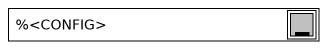
[picture p166: DIGOUT_TOUCH_SMAL (HMI screen)]
rectangle at (0,0)-(311,33): taps $Station$.$Output$
rounded rectangle at (1,1)-(280,32): text "%<CONFIG>"; shows '$Output$'; taps $Station$.$Output$; dynamic style $OutputLocked$
rounded rectangle at (279,2)-(308,31): alarm colour if $OutputLocked$; taps $Station$.$Output$; dynamic style $OutputLocked$
rounded rectangle at (282,5)-(305,28): alarm colour if $Station$.$Output$; taps $Station$.$Output$; tooltip $Output$; dynamic style $OutputLocked$
rectangle at (287,24)-(301,28): invisible if $Station$.$Output$; taps $Station$.$Output$; dynamic style gi16_betriebsart <> HAND
*)

(* Visualisation PRUEFTEILEN_CZ
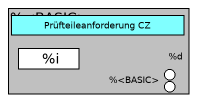
rectangle at (0,0)-(181,86): text "%<BASIC>"; shows 'auto_Prüfteileanforderung'
rectangle at (156,37)-(179,59): text "%d"; shows ST03_Main.CTR; invisible if gTakeTestParts=FALSE AND gTakeTestPartsAuto=FALSE; alarm colour if gTakeTestParts OR gTakeTestPartsAuto
rectangle at (18,61)-(153,82): text "%<BASIC>"; shows 'Rutsche belegt'; invisible if .TD.TestpartBilister
ellipse at (156,61)-(167,72): invisible if .TD.TestpartBilister; alarm colour if ST03_8_75_B13_5.BitInToCheck
ellipse at (156,73)-(167,84): invisible if .TD.TestpartBilister; alarm colour if ST03_8_75_B13_6.BitInToCheck
rectangle at (3,7)-(176,27): text "Prüfteileanforderung CZ"; invisible if TRUE
rectangle at (10,40)-(71,61): text "%i"; shows gPartsTestVisu; editable 0..; dynamic style .ST_CPU.LNG <> 2
*)

(* Visualisation PRUEFTEILEN_DE
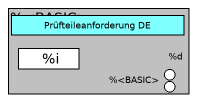
rectangle at (0,0)-(181,86): text "%<BASIC>"; shows 'Prüfteileanforderung'
rectangle at (156,37)-(179,59): text "%d"; shows ST03_Main.CTR; invisible if gTakeTestParts=FALSE AND gTakeTestPartsAuto=FALSE; alarm colour if gTakeTestParts OR gTakeTestPartsAuto
rectangle at (19,61)-(153,82): text "%<BASIC>"; shows 'Rutsche belegt'; invisible if .TD.TestpartBilister
ellipse at (156,61)-(167,72): invisible if .TD.TestpartBilister; alarm colour if ST03_8_75_B13_5.BitInToCheck
ellipse at (156,73)-(167,84): invisible if .TD.TestpartBilister; alarm colour if ST03_8_75_B13_6.BitInToCheck
rectangle at (3,7)-(176,27): text "Prüfteileanforderung DE"; invisible if TRUE
rectangle at (10,40)-(71,61): text "%i"; shows MP.ST03.NoOfTestParts; editable 0..50; dynamic style .ST_CPU.LNG = 2
*)

(* Visualisation PRUEFTEILENTNAHME
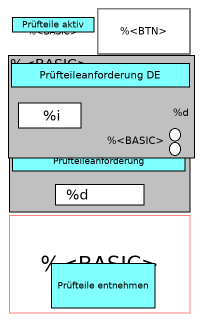
embedded screen at (89,5)-(182,51): ZLIB_VISUBUTTON_S24
rectangle at (1,8)-(88,49): text "%<BASIC>"; shows 'Prüfteile aktiv'; invisible if NOT gTakeTestParts AND NOT gTakeTestPartsAuto; alarm colour if gTakeTestParts OR gTakeTestPartsAuto
rectangle at (1,212)-(182,310): text "%<BASIC>"; shows 'Prüfteile entnehmen'; invisible if NOT ST03_Main.TestPartsRemove; taps gTakeTestPartsFinished
rectangle at (43,260)-(147,305): text "Prüfteile entnehmen"; invisible if TRUE
rectangle at (4,14)-(86,29): text "Prüfteile aktiv"; invisible if TRUE
rectangle at (1,141)-(182,209): text "%<BASIC>"; shows 'Teile seit letzten Test'
rectangle at (4,148)-(177,168): text "Prüfteileanforderung"; invisible if TRUE
rectangle at (47,181)-(136,202): text "%d"; shows gPartsTest; editable 0..1
embedded screen at (0,52)-(187,155): PRUEFTEILEN_CZ
embedded screen at (0,52)-(187,155): PRUEFTEILEN_DE; invisible if .ST_CPU.LNG = 2; dynamic style .ST_CPU.LNG = 2
*)

(* Visualisation ZLIB_SENSOPART
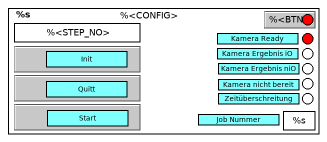
rectangle at (0,0)-(311,126): text "%s"; shows '$FB$'
rectangle at (178,21)-(289,40): text "%<BASIC>"; shows 'Kamera Ready'
rectangle at (178,36)-(289,55): text "%<BASIC>"; shows 'Kamera Ergebnis iO'
rectangle at (178,51)-(289,70): text "%<BASIC>"; shows 'Kamera Ergebnis niO'
rectangle at (6,15)-(132,34): text "%<STEP_NO>"; shows $FB$.fb_state_entry.i16_step; alarm colour if $FB$.fb_state_entry.i16_step=1000
ellipse at (294,25)-(305,36): alarm colour if $FB$.b_ready
ellipse at (294,40)-(305,51): alarm colour if $FB$.Ergebnis_IO
ellipse at (294,55)-(305,66): alarm colour if $FB$.Ergebnis_NIO
rectangle at (178,66)-(289,85): text "%<BASIC>"; shows 'Kamera nicht betriebsbereit'
ellipse at (294,70)-(305,81): alarm colour if $FB$.sm_kamera_nicht_bb
rectangle at (178,81)-(289,100): text "%<BASIC>"; shows 'Zeitüberschreitung'
ellipse at (294,85)-(305,96): alarm colour if $FB$.sm_zeitueberschreitung
rectangle at (155,104)-(266,123): text "%<BASIC>"; shows 'Job Nummer'
rectangle at (275,103)-(307,122): text "%s"; shows $FB$.i16_job; editable 1..4
button at (6,38)-(132,64): text "%<BTN>"; shows 'Init'; dynamic style Color.grey, TRUE
button at (6,67)-(132,93): text "%<BTN>"; shows 'Quitt'; dynamic style Color.grey, TRUE
button at (6,38)-(132,64): text "%<BTN>"; shows 'Init'; invisible if ( *ModeSelect.Mode<>MODE_MANUAL* ); taps $FB$.b_init; dynamic style Color.lightgrey, Color.grey, ( *ModeSelect.Mode<>MODE_MANUAL* )
button at (6,67)-(132,93): text "%<BTN>"; shows 'Quitt'; invisible if ( *ModeSelect.Mode<>MODE_MANUAL* ); taps $FB$.b_quitt; dynamic style Color.lightgrey, Color.grey, ( *ModeSelect.Mode<>MODE_MANUAL* )
button at (6,96)-(132,122): text "%<BTN>"; shows 'Start'; dynamic style Color.grey, TRUE
button at (6,96)-(132,122): text "%<BTN>"; shows 'Start'; invisible if ( *ModeSelect.Mode<>MODE_MANUAL* ); taps $FB$.b_start_manual; dynamic style Color.lightgrey, Color.grey, ( *ModeSelect.Mode<>MODE_MANUAL* )
button at (256,3)-(307,20): text "%<BTN>"; shows MP.ST00.IFMCameraActiveText; toggles $Cam_On$; dynamic style color.lightgrey, TRUE
ellipse at (294,6)-(305,17): alarm colour if $Cam_On$
rectangle at (110,1)-(240,14): text "%<CONFIG>"; shows '$FB$'
rectangle at (209,25)-(290,36): text "Kamera Ready"; invisible if TRUE
rectangle at (209,40)-(290,51): text "Kamera Ergebnis iO"; invisible if TRUE
rectangle at (210,55)-(291,66): text "Kamera Ergebnis niO"; invisible if TRUE
rectangle at (210,71)-(291,82): text "Kamera nicht bereit"; invisible if TRUE
rectangle at (210,85)-(291,96): text "Zeitüberschreitung"; invisible if TRUE
rectangle at (190,106)-(271,117): text "Job Nummer"; invisible if TRUE
rectangle at (39,102)-(120,118): text "Start"; invisible if TRUE
rectangle at (38,73)-(119,89): text "Quitt"; invisible if TRUE
rectangle at (38,43)-(119,59): text "Init"; invisible if TRUE
*)

(* Visualisation ZLIB_SENSOPART_1
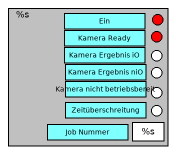
rectangle at (0,0)-(160,138): text "%s"; shows '$FB$'
rectangle at (27,17)-(138,36): text "%<BASIC>"; shows 'Kamera Ready'
rectangle at (27,37)-(138,56): text "%<BASIC>"; shows 'Kamera Ergebnis iO'
rectangle at (27,54)-(138,73): text "%<BASIC>"; shows 'Kamera Ergebnis niO'
ellipse at (143,23)-(154,34): alarm colour if $FB$.b_ready
ellipse at (143,42)-(154,53): alarm colour if $FB$.Ergebnis_IO
ellipse at (143,59)-(154,70): alarm colour if $FB$.Ergebnis_NIO
rectangle at (3,73)-(140,92): text "%<BASIC>"; shows 'Kamera nicht betriebsbereit'
ellipse at (143,79)-(154,90): alarm colour if $FB$.sm_kamera_nicht_bb
rectangle at (27,92)-(138,111): text "%<BASIC>"; shows 'Zeitüberschreitung'
ellipse at (143,97)-(154,108): alarm colour if $FB$.sm_zeitueberschreitung
rectangle at (10,114)-(121,133): text "%<BASIC>"; shows 'Job Nummer'
rectangle at (124,114)-(156,133): text "%s"; shows $FB$.i16_job
ellipse at (144,6)-(155,17): alarm colour if $Cam_On$
rectangle at (113,2)-(139,21): text "%<BASIC>"; shows 'Ein'
rectangle at (56,5)-(137,21): text "Ein"; invisible if TRUE
rectangle at (56,22)-(137,38): text "Kamera Ready"; invisible if TRUE
rectangle at (56,39)-(137,55): text "Kamera Ergebnis iO"; invisible if TRUE
rectangle at (57,56)-(138,72): text "Kamera Ergebnis niO"; invisible if TRUE
rectangle at (57,73)-(138,89): text "Kamera nicht betriebsbereit"; invisible if TRUE
rectangle at (57,94)-(138,110): text "Zeitüberschreitung"; invisible if TRUE
rectangle at (39,116)-(120,132): text "Job Nummer"; invisible if TRUE
*)

(* Visualisation ZLIB_SENSOPART_2
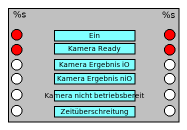
rectangle at (0,0)-(171,114): text "%s"; shows '$FB1$'
ellipse at (156,36)-(167,47): alarm colour if $FB2$.b_ready
ellipse at (156,51)-(167,62): alarm colour if $FB2$.Ergebnis_IO
ellipse at (156,65)-(167,76): alarm colour if $FB2$.Ergebnis_NIO
ellipse at (156,81)-(167,92): alarm colour if $FB2$.sm_kamera_nicht_bb
ellipse at (156,97)-(167,108): alarm colour if $FB2$.sm_zeitueberschreitung
ellipse at (156,21)-(167,32): alarm colour if $Cam_On2$
ellipse at (3,36)-(14,47): alarm colour if $FB1$.b_ready
ellipse at (3,51)-(14,62): alarm colour if $FB1$.Ergebnis_IO
ellipse at (3,65)-(14,76): alarm colour if $FB1$.Ergebnis_NIO
ellipse at (3,81)-(14,92): alarm colour if $FB1$.sm_kamera_nicht_bb
ellipse at (3,97)-(14,108): alarm colour if $FB1$.sm_zeitueberschreitung
ellipse at (3,21)-(14,32): alarm colour if $Cam_On1$
rectangle at (85,0)-(169,14): text "%s"; shows '$FB2$'
rectangle at (17,31)-(154,50): text "%<BASIC>"; shows 'Kamera Ready'
rectangle at (17,47)-(154,66): text "%<BASIC>"; shows 'Kamera Ergebnis iO'
rectangle at (17,61)-(154,80): text "%<BASIC>"; shows 'Kamera Ergebnis niO'
rectangle at (17,77)-(154,96): text "%<BASIC>"; shows 'Kamera nicht betriebsbereit'
rectangle at (17,93)-(154,112): text "%<BASIC>"; shows 'Zeitüberschreitung'
rectangle at (17,18)-(154,37): text "%<BASIC>"; shows 'Ein'
rectangle at (46,22)-(127,33): text "Ein"; invisible if TRUE
rectangle at (46,35)-(127,46): text "Kamera Ready"; invisible if TRUE
rectangle at (46,51)-(127,62): text "Kamera Ergebnis iO"; invisible if TRUE
rectangle at (46,65)-(127,76): text "Kamera Ergebnis niO"; invisible if TRUE
rectangle at (46,82)-(127,93): text "Kamera nicht betriebsbereit"; invisible if TRUE
rectangle at (46,98)-(127,109): text "Zeitüberschreitung"; invisible if TRUE
*)

(* Visualisation ZLIB_SENSOPART_3
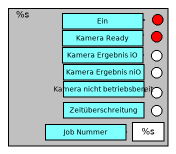
rectangle at (0,0)-(160,138): text "%s"; shows '$FB$'
ellipse at (143,23)-(154,34): alarm colour if $FB$.b_ready
ellipse at (143,42)-(154,53): alarm colour if $FB$.Ergebnis_IO
ellipse at (143,59)-(154,70): alarm colour if $FB$.Ergebnis_NIO
ellipse at (143,79)-(154,90): alarm colour if $FB$.sm_kamera_nicht_bb
ellipse at (143,97)-(154,108): alarm colour if $FB$.sm_zeitueberschreitung
rectangle at (124,114)-(156,133): text "%s"; shows $FB$.i16_job
ellipse at (144,6)-(155,17): alarm colour if $Cam_On$
rectangle at (28,17)-(139,36): text "%<BASIC>"; shows 'Kamera Ready'
rectangle at (28,37)-(139,56): text "%<BASIC>"; shows 'Kamera Ergebnis iO'
rectangle at (28,54)-(139,73): text "%<BASIC>"; shows 'Kamera Ergebnis niO'
rectangle at (4,73)-(141,92): text "%<BASIC>"; shows 'Kamera nicht betriebsbereit'
rectangle at (28,92)-(139,111): text "%<BASIC>"; shows 'Zeitüberschreitung'
rectangle at (11,114)-(122,133): text "%<BASIC>"; shows 'Job Nummer'
rectangle at (114,2)-(140,21): text "%<BASIC>"; shows 'Ein'
rectangle at (54,5)-(135,21): text "Ein"; invisible if TRUE
rectangle at (54,22)-(135,38): text "Kamera Ready"; invisible if TRUE
rectangle at (54,39)-(135,55): text "Kamera Ergebnis iO"; invisible if TRUE
rectangle at (55,56)-(136,72): text "Kamera Ergebnis niO"; invisible if TRUE
rectangle at (55,73)-(136,89): text "Kamera nicht betriebsbereit"; invisible if TRUE
rectangle at (55,94)-(136,110): text "Zeitüberschreitung"; invisible if TRUE
rectangle at (37,116)-(118,132): text "Job Nummer"; invisible if TRUE
*)

(* Visualisation ZLIB_SENSOPART_4
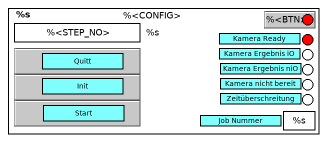
rectangle at (0,0)-(311,126): text "%s"; shows '$FB$'
rectangle at (6,15)-(132,34): text "%<STEP_NO>"; shows $FB$.fb_state_entry.i16_step; alarm colour if $FB$.fb_state_entry.i16_step=1000
ellipse at (294,26)-(305,37): alarm colour if $FB$.st_ctrl_out.b_bereit
ellipse at (294,41)-(305,52): alarm colour if $FB$.b_Kam_Pruef_IO
ellipse at (294,56)-(305,67): alarm colour if $FB$.b_Kam_Pruef_NIO
ellipse at (294,71)-(305,82): alarm colour if $FB$.sm_kamera_nicht_bb
ellipse at (294,86)-(305,97): alarm colour if $FB$.sm_kamera_keine_reaktion
rectangle at (275,103)-(307,122): text "%s"; shows $FB$.JobNo; editable 1..4
button at (6,66)-(132,92): text "%<BTN>"; shows 'Init'; dynamic style Color.grey, TRUE
button at (6,40)-(132,66): text "%<BTN>"; shows 'Quitt'; dynamic style Color.grey, TRUE
button at (6,66)-(132,92): text "%<BTN>"; shows 'Init'; invisible if ModeSelect.Mode<>MODE_MANUAL; taps $FB$.st_ctrl_in.b_init; dynamic style Color.lightgrey, Color.grey
button at (6,40)-(132,66): text "%<BTN>"; shows 'Quitt'; invisible if ModeSelect.Mode<>MODE_MANUAL; taps $FB$.st_ctrl_in.b_quitt; dynamic style Color.lightgrey, Color.grey
button at (6,92)-(132,118): text "%<BTN>"; shows 'Start'; dynamic style Color.grey, TRUE
button at (6,92)-(132,118): text "%<BTN>"; shows 'Start'; invisible if ModeSelect.Mode<>MODE_MANUAL; taps $FB$.st_ctrl_in.b_start; dynamic style Color.lightgrey, Color.grey
button at (256,3)-(307,20): text "%<BTN>"; shows MP.ST00.IFMCameraActiveText; toggles $Cam_On$; dynamic style color.lightgrey, FALSE
ellipse at (294,6)-(305,17): alarm colour if $Cam_On$
rectangle at (107,1)-(246,14): text "%<CONFIG>"; shows '$FB$'
rectangle at (35,97)-(116,113): text "Start"; invisible if TRUE
rectangle at (34,45)-(115,61): text "Quitt"; invisible if TRUE
rectangle at (34,70)-(115,86): text "Init"; invisible if TRUE
rectangle at (179,22)-(290,41): text "%<BASIC>"; shows 'Kamera Ready'
rectangle at (179,37)-(290,56): text "%<BASIC>"; shows 'Kamera Ergebnis iO'
rectangle at (179,52)-(290,71): text "%<BASIC>"; shows 'Kamera Ergebnis niO'
rectangle at (179,67)-(290,86): text "%<BASIC>"; shows 'Kamera nicht betriebsbereit'
rectangle at (179,82)-(290,101): text "%<BASIC>"; shows 'Zeitüberschreitung'
rectangle at (159,104)-(270,123): text "%<BASIC>"; shows 'Job Nummer'
rectangle at (211,25)-(292,36): text "Kamera Ready"; invisible if TRUE
rectangle at (211,40)-(292,51): text "Kamera Ergebnis iO"; invisible if TRUE
rectangle at (212,55)-(293,66): text "Kamera Ergebnis niO"; invisible if TRUE
rectangle at (212,70)-(293,81): text "Kamera nicht bereit"; invisible if TRUE
rectangle at (212,85)-(293,96): text "Zeitüberschreitung"; invisible if TRUE
rectangle at (192,107)-(273,118): text "Job Nummer"; invisible if TRUE
rectangle at (133,15)-(214,34): text "%s"; shows $FB$.RecvDataString
*)

(* Visualisation ZLIB_SENSOPART_4_2
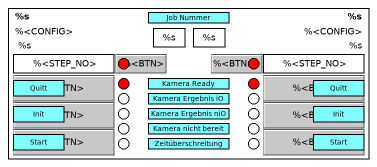
rectangle at (5,46)-(106,65): text "%<STEP_NO>"; shows $FB$.fb_state_entry.i16_step; alarm colour if $FB$.fb_state_entry.i16_step=1000
ellipse at (240,70)-(251,81): alarm colour if $FB2$.st_ctrl_out.b_bereit
ellipse at (240,85)-(251,96): alarm colour if $FB2$.b_Kam_Pruef_IO
ellipse at (240,100)-(251,111): alarm colour if $FB2$.b_Kam_Pruef_NIO
ellipse at (240,115)-(251,126): alarm colour if $FB2$.sm_kamera_nicht_bb
ellipse at (240,130)-(251,141): alarm colour if $FB2$.sm_zeitueberschreitung
rectangle at (145,20)-(177,39): text "%s"; shows $FB$.JobNo; editable 1..4
button at (5,94)-(106,120): text "%<BTN>"; shows 'Init'; dynamic style Color.grey, TRUE
button at (5,94)-(106,120): text "%<BTN>"; shows 'Init'; invisible if ModeSelect.Mode<>MODE_MANUAL; taps $FB$.st_ctrl_in.b_init; dynamic style Color.lightgrey, Color.grey
button at (5,67)-(106,93): text "%<BTN>"; shows 'Quitt'; dynamic style Color.grey, TRUE
button at (5,67)-(106,93): text "%<BTN>"; shows 'Quitt'; invisible if ModeSelect.Mode<>MODE_MANUAL; taps $FB$.st_ctrl_in.b_quitt; dynamic style Color.lightgrey, Color.grey
button at (5,121)-(106,147): text "%<BTN>"; shows 'Start'; dynamic style Color.grey, TRUE
button at (5,121)-(106,147): text "%<BTN>"; shows 'Start'; invisible if ModeSelect.Mode<>MODE_MANUAL; taps $FB$.st_ctrl_in.b_start; dynamic style Color.lightgrey, Color.grey
button at (203,46)-(254,65): text "%<BTN>"; shows MP.ST00.IFMCameraActiveText; toggles $Cam_On2$; dynamic style color.lightgrey, FALSE
ellipse at (240,50)-(251,61): alarm colour if $Cam_On2$
rectangle at (5,17)-(144,30): text "%<CONFIG>"; shows '$FB$'
rectangle at (5,126)-(56,142): text "Start"; invisible if TRUE
rectangle at (5,72)-(56,88): text "Quitt"; invisible if TRUE
rectangle at (5,98)-(56,114): text "Init"; invisible if TRUE
rectangle at (125,66)-(236,85): text "%<BASIC>"; shows 'Kamera Ready'
rectangle at (125,81)-(236,100): text "%<BASIC>"; shows 'Kamera Ergebnis iO'
rectangle at (125,96)-(236,115): text "%<BASIC>"; shows 'Kamera Ergebnis niO'
rectangle at (125,111)-(236,130): text "%<BASIC>"; shows 'Kamera nicht betriebsbereit'
rectangle at (125,126)-(236,145): text "%<BASIC>"; shows 'Zeitüberschreitung'
rectangle at (125,2)-(236,15): text "%<BASIC>"; shows 'Job Nummer'
rectangle at (140,70)-(221,81): text "Kamera Ready"; invisible if TRUE
rectangle at (140,85)-(221,96): text "Kamera Ergebnis iO"; invisible if TRUE
rectangle at (140,100)-(221,111): text "Kamera Ergebnis niO"; invisible if TRUE
rectangle at (140,115)-(221,126): text "Kamera nicht bereit"; invisible if TRUE
rectangle at (140,130)-(221,141): text "Zeitüberschreitung"; invisible if TRUE
rectangle at (140,4)-(221,15): text "Job Nummer"; invisible if TRUE
rectangle at (5,31)-(86,44): text "%s"; shows $FB$.RecvDataString
ellipse at (110,70)-(121,81): alarm colour if $FB$.st_ctrl_out.b_bereit
ellipse at (110,85)-(121,96): alarm colour if $FB$.b_Kam_Pruef_IO
ellipse at (110,100)-(121,111): alarm colour if $FB$.b_Kam_Pruef_NIO
ellipse at (110,115)-(121,126): alarm colour if $FB$.sm_kamera_nicht_bb
ellipse at (110,130)-(121,141): alarm colour if $FB$.sm_zeitueberschreitung
button at (107,46)-(158,65): text "%<BTN>"; shows MP.ST00.IFMCameraActiveText; toggles $Cam_On$; dynamic style color.lightgrey, FALSE
ellipse at (110,50)-(121,61): alarm colour if $Cam_On$
rectangle at (5,2)-(144,15): text "%s"; shows '$FB$'
rectangle at (217,17)-(356,30): text "%<CONFIG>"; shows '$FB2$'
rectangle at (217,2)-(356,15): text "%s"; shows '$FB2$'
rectangle at (275,31)-(356,44): text "%s"; shows $FB2$.RecvDataString
rectangle at (255,46)-(356,65): text "%<STEP_NO>"; shows $FB2$.fb_state_entry.i16_step; alarm colour if $FB2$.fb_state_entry.i16_step=1000
button at (255,94)-(356,120): text "%<BTN>"; shows 'Init'; dynamic style Color.grey, TRUE
button at (255,94)-(356,120): text "%<BTN>"; shows 'Init'; invisible if ModeSelect.Mode<>MODE_MANUAL; taps $FB2$.st_ctrl_in.b_init; dynamic style Color.lightgrey, Color.grey
button at (255,67)-(356,93): text "%<BTN>"; shows 'Quitt'; dynamic style Color.grey, TRUE
button at (255,67)-(356,93): text "%<BTN>"; shows 'Quitt'; invisible if ModeSelect.Mode<>MODE_MANUAL; taps $FB2$.st_ctrl_in.b_quitt; dynamic style Color.lightgrey, Color.grey
button at (255,121)-(356,147): text "%<BTN>"; shows 'Start'; dynamic style Color.grey, TRUE
button at (255,121)-(356,147): text "%<BTN>"; shows 'Start'; invisible if ModeSelect.Mode<>MODE_MANUAL; taps $FB2$.st_ctrl_in.b_start; dynamic style Color.lightgrey, Color.grey
rectangle at (305,126)-(356,142): text "Start"; invisible if TRUE
rectangle at (305,72)-(356,88): text "Quitt"; invisible if TRUE
rectangle at (305,98)-(356,114): text "Init"; invisible if TRUE
rectangle at (185,20)-(217,39): text "%s"; shows $FB2$.JobNo; editable 1..4
1 more shapes without text or variables
*)

(* Visualisation ZLIB_SENSOPART_5
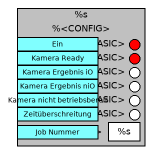
rectangle at (0,0)-(128,138): text "%s"; shows '$FB$'
rectangle at (2,40)-(110,59): text "%<BASIC>"; shows 'Kamera Ready'
rectangle at (2,54)-(110,73): text "%<BASIC>"; shows 'Kamera Ergebnis iO'
rectangle at (2,68)-(110,87): text "%<BASIC>"; shows 'Kamera Ergebnis niO'
rectangle at (2,96)-(110,115): text "%<BASIC>"; shows 'Zeitüberschreitung'
rectangle at (2,114)-(87,133): text "%<BASIC>"; shows 'Job Nummer'
rectangle at (91,114)-(123,133): text "%s"; shows $FB$.JobNo
ellipse at (112,31)-(123,42): alarm colour if $Cam_On$
rectangle at (2,26)-(110,45): text "%<BASIC>"; shows 'Ein'
rectangle at (0,29)-(81,43): text "Ein"; invisible if TRUE
rectangle at (0,117)-(81,131): text "Job Nummer"; invisible if TRUE
ellipse at (112,45)-(123,56): alarm colour if $FB$.st_ctrl_out.b_bereit
ellipse at (112,59)-(123,70): alarm colour if $FB$.b_Kam_Pruef_IO
ellipse at (112,73)-(123,84): alarm colour if $FB$.b_Kam_Pruef_NIO
ellipse at (112,87)-(123,98): alarm colour if $FB$.sm_kamera_nicht_bb
ellipse at (112,101)-(123,112): alarm colour if $FB$.sm_zeitueberschreitung
rectangle at (0,43)-(81,57): text "Kamera Ready"; invisible if TRUE
rectangle at (0,57)-(81,71): text "Kamera Ergebnis iO"; invisible if TRUE
rectangle at (0,71)-(81,85): text "Kamera Ergebnis niO"; invisible if TRUE
rectangle at (0,99)-(81,113): text "Zeitüberschreitung"; invisible if TRUE
rectangle at (2,82)-(110,101): text "%<BASIC>"; shows 'Kamera nicht betriebsbereit'
rectangle at (0,85)-(81,99): text "Kamera nicht betriebsbereit"; invisible if TRUE
rectangle at (2,14)-(126,27): text "%<CONFIG>"; shows '$FB$'
*)

(* Visualisation ZLIB_SENSOPART_6
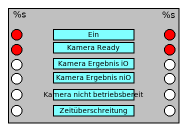
rectangle at (0,0)-(171,115): text "%s"; shows '$FB1$'
rectangle at (16,30)-(153,49): text "%<BASIC>"; shows 'Kamera Ready'
rectangle at (16,46)-(153,65): text "%<BASIC>"; shows 'Kamera Ergebnis iO'
rectangle at (16,60)-(153,79): text "%<BASIC>"; shows 'Kamera Ergebnis niO'
ellipse at (156,36)-(167,47): alarm colour if $FB2$.st_ctrl_out.b_bereit
ellipse at (156,51)-(167,62): alarm colour if $FB2$.b_Kam_Pruef_IO
ellipse at (156,65)-(167,76): alarm colour if $FB2$.b_Kam_Pruef_NIO
rectangle at (16,76)-(153,95): text "%<BASIC>"; shows 'Kamera nicht betriebsbereit'
ellipse at (156,81)-(167,92): alarm colour if $FB2$.sm_kamera_nicht_bb
rectangle at (16,92)-(153,111): text "%<BASIC>"; shows 'Zeitüberschreitung'
ellipse at (156,97)-(167,108): alarm colour if $FB2$.sm_zeitueberschreitung
ellipse at (156,21)-(167,32): alarm colour if $Cam_On2$
rectangle at (16,17)-(153,36): text "%<BASIC>"; shows 'Ein'
ellipse at (3,36)-(14,47): alarm colour if $FB1$.st_ctrl_out.b_bereit
ellipse at (3,51)-(14,62): alarm colour if $FB1$.b_Kam_Pruef_IO
ellipse at (3,65)-(14,76): alarm colour if $FB1$.b_Kam_Pruef_NIO
ellipse at (3,81)-(14,92): alarm colour if $FB1$.sm_kamera_nicht_bb
ellipse at (3,97)-(14,108): alarm colour if $FB1$.sm_zeitueberschreitung
ellipse at (3,21)-(14,32): alarm colour if $Cam_On1$
rectangle at (85,0)-(169,14): text "%s"; shows '$FB2$'
rectangle at (45,21)-(126,32): text "Ein"; invisible if TRUE
rectangle at (45,34)-(126,45): text "Kamera Ready"; invisible if TRUE
rectangle at (45,50)-(126,61): text "Kamera Ergebnis iO"; invisible if TRUE
rectangle at (45,64)-(126,75): text "Kamera Ergebnis niO"; invisible if TRUE
rectangle at (45,81)-(126,92): text "Kamera nicht betriebsbereit"; invisible if TRUE
rectangle at (45,97)-(126,108): text "Zeitüberschreitung"; invisible if TRUE
*)

(* Visualisation ZLIB_SENSOPART_7
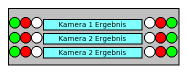
rectangle at (34,5)-(134,24): text "%<BASIC>"; shows 'Kamera 1 Ergebnis'
rectangle at (34,19)-(134,38): text "%<BASIC>"; shows 'Kamera 2 Ergebnis'
ellipse at (147,24)-(158,35): alarm colour if $FB2$.st_ctrl_out.b_bereit
ellipse at (136,9)-(147,20): alarm colour if $FB2$.b_Kam_Pruef_IO
ellipse at (136,24)-(147,35): alarm colour if $FB2$.b_Kam_Pruef_NIO
ellipse at (136,38)-(147,49): alarm colour if $FB2$.sm_kamera_nicht_bb
ellipse at (147,9)-(158,20): alarm colour if $Cam_On2$
ellipse at (12,24)-(23,35): alarm colour if $FB1$.st_ctrl_out.b_bereit
ellipse at (23,9)-(34,20): alarm colour if $FB1$.b_Kam_Pruef_IO
ellipse at (23,24)-(34,35): alarm colour if $FB1$.b_Kam_Pruef_NIO
ellipse at (23,38)-(34,49): alarm colour if $FB1$.sm_kamera_nicht_bb
ellipse at (12,9)-(23,20): alarm colour if $Cam_On1$
rectangle at (34,33)-(134,52): text "%<BASIC>"; shows 'Kamera 3 Ergebnis'
ellipse at (147,38)-(158,49): alarm colour if $FB2$.st_ctrl_out.b_bereit
ellipse at (12,38)-(23,49): alarm colour if $FB1$.st_ctrl_out.b_bereit
ellipse at (158,24)-(169,35): alarm colour if $FB2$.st_ctrl_out.b_bereit
ellipse at (158,9)-(169,20): alarm colour if $Cam_On2$
ellipse at (158,38)-(169,49): alarm colour if $FB2$.st_ctrl_out.b_bereit
ellipse at (1,24)-(12,35): alarm colour if $FB2$.st_ctrl_out.b_bereit
ellipse at (1,9)-(12,20): alarm colour if $Cam_On2$
ellipse at (1,38)-(12,49): alarm colour if $FB2$.st_ctrl_out.b_bereit
rectangle at (35,11)-(134,22): text "Kamera 1 Ergebnis"; invisible if TRUE
rectangle at (35,25)-(134,36): text "Kamera 2 Ergebnis"; invisible if TRUE
rectangle at (35,39)-(134,50): text "Kamera 2 Ergebnis"; invisible if TRUE
1 more shapes without text or variables
*)

(* Visualisation SIGNS_PUMP
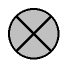
ellipse at (0,0)-(51,51): alarm colour if $Object$.BitOutToSet; taps $Object$.Pressed; dynamic style NOT $Object$.Enable
polyline at (8,8)-(43,43): alarm colour if NOT $Object$.Enable; taps $Object$.Pressed; angle $Pos$/4; dynamic style NOT $Object$.Enable
polyline at (8,8)-(43,43): alarm colour if NOT $Object$.Enable; taps $Object$.Pressed; angle $Pos$/4; dynamic style NOT $Object$.Enable
*)

(* Visualisation ZLIB_TIPPL
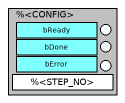
rectangle at (0,0)-(109,87): text "%<CONFIG>"; shows '$Objekt$'
rectangle at (5,27)-(87,46): text "%<BASIC>"; shows 'bDone'
rectangle at (5,47)-(87,66): text "%<BASIC>"; shows 'bError'
ellipse at (92,33)-(103,44): alarm colour if $Objekt$.bDone
ellipse at (92,52)-(103,63): alarm colour if $Objekt$.bError
ellipse at (92,16)-(103,27): alarm colour if $Objekt$.bReady
rectangle at (5,12)-(88,31): text "%<BASIC>"; shows 'bReady'
rectangle at (8,14)-(89,30): text "bReady"; invisible if TRUE
rectangle at (8,31)-(89,47): text "bDone"; invisible if TRUE
rectangle at (8,48)-(89,64): text "bError"; invisible if TRUE
rectangle at (4,66)-(105,82): text "%<STEP_NO>"; shows $Objekt$.fb_state_entry.i16_step; alarm colour if $Objekt$.fb_state_entry.i16_step = FEHLER
rectangle at (4,66)-(105,82): text "%<STEP_NO>"; shows $Objekt$.fb_state_entry.i16_step; invisible if $Objekt$.fb_state_entry.i16_step >= 980; alarm colour if $Objekt$.fb_state_entry.i16_step = 100
*)

(* Visualisation ZUFUEHRUNG
rectangle at (0,0)-(524,482): invisible if TRUE
rectangle at (464,405)-(513,466): text "Roboter"; invisible if TRUE; opens MANUAL_ST03_0
rectangle at (7,2)-(274,318): text "Zähler"; invisible if TRUE; opens MANUAL_ST03_0
button at (7,402)-(119,453): text "%<BTN>"; shows 'TaktBand'; invisible if gTypeCode<>4991 AND gTypeCode <>312; taps ST03_Band.b_MoveRel; dynamic style Color.lightgrey, Color.grey
rectangle at (10,407)-(114,452): text "Takt Förderband"; invisible if TRUE
rectangle at (7,324)-(124,395): text "%<BASIC>"; shows 'Föderband'; invisible if MP.ST03.SGM_3621
embedded screen at (9,338)-(120,392): ZLIB_OVERRIDE; invisible if MP.ST03.SGM_3621
embedded screen at (245,5)-(522,481): ZUFUEHRUNG_93POL; invisible if gTypeCode<>4991 AND gTypeCode <>312
embedded screen at (360,1)-(423,473): ZUFUEHRUNG_92POL; invisible if gTypeCode <>550
embedded screen at (331,9)-(392,480): ZUFUEHRUNG_154RP; invisible if gTypeCode<>4872
embedded screen at (423,7)-(464,483): ZUFUEHRUNG_74_91_168POL; invisible if gTypeCode<>360 AND gTypeCode <>379 AND gTypeCode <>489
embedded screen at (378,8)-(419,480): ZUFUEHRUNG_154POL; invisible if gTypeCode<>4871
embedded screen at (400,0)-(460,481): ZUFUEHRUNG_35POL; invisible if gTypeCode <>4992
embedded screen at (348,5)-(420,477): ZUFUEHRUNG_206POL; invisible if gTypeCode<>522
embedded screen at (368,2)-(440,474): ZUFUEHRUNG_124POL; invisible if gTypeCode<>564
embedded screen at (332,3)-(483,475): ZUFUEHRUNG_46POL; invisible if gTypeCode<>569
embedded screen at (142,6)-(496,473): ZUFUEHRUNG_NOX_5_6POL; invisible if gTypeCode<>5632  AND gTypeCode<>5633
embedded screen at (250,5)-(491,477): ZUFUEHRUNG_NOX_4POL; invisible if gTypeCode<>5631
embedded screen at (390,8)-(462,480): ZUFUEHRUNG_88POL; invisible if gTypeCode<>5731
embedded screen at (394,7)-(487,478): ZUFUEHRUNG_7POL; invisible if gTypeCode<>575  AND gTypeCode<>5753  AND gTypeCode<>5754  AND gTypeCode<>5755
embedded screen at (409,10)-(479,482): ZUFUEHRUNG_88POL_AMG; invisible if gTypeCode<>5732
embedded screen at (404,10)-(474,482): ZUFUEHRUNG_120POL; invisible if gTypeCode<>5771
embedded screen at (399,10)-(469,482): ZUFUEHRUNG_21POL; invisible if gTypeCode<>5772
embedded screen at (394,10)-(464,482): ZUFUEHRUNG_191POL; invisible if gTypeCode<>580
embedded screen at (363,1)-(433,477): ZUFUEHRUNG_72POL; invisible if gTypeCode<>5831
embedded screen at (365,6)-(435,477): ZUFUEHRUNG_48POL; invisible if gTypeCode<>5832
embedded screen at (328,3)-(510,479): ZUFUEHRUNG_268POL_RP; invisible if gTypeCode<>5842
embedded screen at (262,7)-(518,484): ZUFUEHRUNG_268POL_102POL_NEU; invisible if gTypeCode<>5841 AND gTypeCode<>4993
embedded screen at (404,7)-(488,478): ZUFUEHRUNG_33POL; invisible if gTypeCode<>598
*)

(* Visualisation ZUFUEHRUNG_120POL
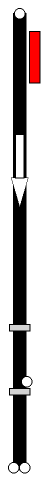
embedded screen at (9,126)-(26,199): SIGNS_ARROWDOWN
ellipse at (12,0)-(23,11): alarm colour if ST03_531_B69_0.BitInToCheck; tooltip ST03_531_B69_0
ellipse at (19,368)-(30,379): alarm colour if ST03_531_B69_6.BitInToCheck; tooltip ST03_531_B69_6
rectangle at (7,380)-(28,387): alarm colour if ST03_531_B69_4.ValveSensor; tooltip ST03_531_B69_3
rectangle at (7,316)-(28,323): alarm colour if ST03_531_B69_2.ValveSensor; tooltip ST03_531_B69_1
rounded rectangle at (27,23)-(38,75): alarm colour if ST03_Init_Lockings.b_freiFuerSG; tooltip b_freiFuerSG
ellipse at (17,454)-(28,465): alarm colour if ST03_531_B69_7.BitInToCheck; tooltip ST03_531_B69_7
ellipse at (6,454)-(17,465): alarm colour if ST03_532_B70_0.BitInToCheck; tooltip ST03_532_B70_0
2 more shapes without text or variables
*)

(* Visualisation ZUFUEHRUNG_124POL
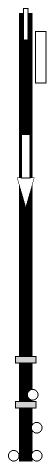
ellipse at (10,447)-(21,458): alarm colour if ST03_452_B70_1.BitInToCheck; tooltip ST03_452_B70_1
embedded screen at (19,131)-(36,204): SIGNS_ARROWDOWN
ellipse at (33,419)-(44,430): alarm colour if ST03_452_B70_2.BitInToCheck; tooltip ST03_452_B70_2
ellipse at (33,447)-(44,458): alarm colour if ST03_453_B70_4.BitInToCheck; tooltip ST03_453_B70_4
ellipse at (29,386)-(40,397): alarm colour if ST03_451_B69_7.BitInToCheck; tooltip ST03_451_B69_7
rectangle at (17,398)-(38,405): alarm colour if ST03_451_B69_2.ValveSensor; tooltip ST03_451_B69_2
rectangle at (17,353)-(38,360): alarm colour if ST03_451_B69_1.ValveSensor; tooltip ST03_451_B69_1
rounded rectangle at (37,28)-(48,80): alarm colour if ST03_Init_Lockings.b_freiFuerSG; tooltip b_freiFuerSG
rounded rectangle at (25,5)-(30,37): alarm colour if ST03_451_B69_4.BitInToCheck; tooltip ST03_451_B69_4
1 more shapes without text or variables
*)

(* Visualisation ZUFUEHRUNG_154POL
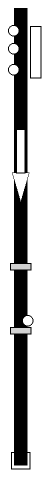
ellipse at (5,35)-(16,46): alarm colour if ST03_425_B67_5.BitInToCheck; tooltip ST03_425_B67_5
embedded screen at (9,121)-(26,194): SIGNS_ARROWDOWN
ellipse at (5,56)-(16,67): alarm colour if ST03_425_B67_6.BitInToCheck; tooltip ST03_425_B67_6
ellipse at (5,17)-(16,28): alarm colour if ST03_425_B67_4.BitInToCheck; tooltip ST03_425_B67_4
ellipse at (19,307)-(30,318): alarm colour if ST03_425_B67_7.BitInToCheck; tooltip ST03_425_B67_7
rectangle at (7,319)-(28,326): alarm colour if ST03_425_B67_2.ValveSensor; tooltip ST03_425_B67_2
rectangle at (7,255)-(28,262): alarm colour if ST03_425_B67_0.ValveSensor; tooltip ST03_425_B67_0
rounded rectangle at (8,444)-(27,461): alarm colour if ST03_426_B68_4.BitInToCheck; tooltip ST03_426_B68_4
rounded rectangle at (27,18)-(38,70): alarm colour if ST03_Init_Lockings.b_freiFuerSG; tooltip b_freiFuerSG
2 more shapes without text or variables
*)

(* Visualisation ZUFUEHRUNG_154RP
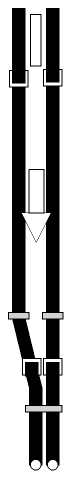
embedded screen at (13,161)-(43,234): SIGNS_ARROWDOWN
ellipse at (39,451)-(50,462): alarm colour if ST03_419_B61_3.BitInToCheck; tooltip ST03_419_B61_3
ellipse at (22,451)-(33,462): alarm colour if ST03_419_B61_2.BitInToCheck; tooltip ST03_419_B61_2
rounded rectangle at (35,350)-(54,367): alarm colour if ST03_419_B61_1.BitInToCheck; tooltip ST03_419_B61_1
rounded rectangle at (14,350)-(33,367): alarm colour if ST03_419_B61_0.BitInToCheck; tooltip ST03_419_B61_0
rectangle at (17,397)-(54,404): alarm colour if ST03_418_B60_5.ValveSensor; tooltip ST03_418_B60_5
rectangle at (0,304)-(21,311): alarm colour if ST03_418_B60_0.ValveSensor; tooltip ST03_418_B60_0
rectangle at (34,304)-(55,311): alarm colour if ST03_418_B60_2.ValveSensor; tooltip ST03_418_B60_2
rounded rectangle at (35,61)-(54,78): alarm colour if ST03_418_B60_7.BitInToCheck; tooltip ST03_418_B60_7
rounded rectangle at (1,62)-(20,79): alarm colour if ST03_418_B60_6.BitInToCheck; tooltip ST03_418_B60_6
rounded rectangle at (22,6)-(33,58): alarm colour if ST03_Init_Lockings.b_freiFuerSG; tooltip b_freiFuerSG
8 more shapes without text or variables
*)

(* Visualisation ZUFUEHRUNG_160POL
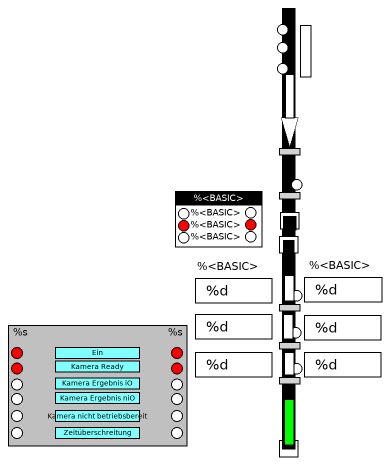
ellipse at (269,34)-(280,45): alarm colour if ST03_421_B63_5.BitInToCheck; tooltip ST03_421_B63_5
embedded screen at (273,66)-(290,139): SIGNS_ARROWDOWN
rounded rectangle at (272,204)-(291,221): alarm colour if ST03_422_B64_0.BitInToCheck; tooltip ST03_422_B64_0
ellipse at (269,55)-(280,66): alarm colour if ST03_421_B63_6.BitInToCheck; tooltip ST03_421_B63_6
ellipse at (269,16)-(280,27): alarm colour if ST03_421_B63_4.BitInToCheck; tooltip ST03_421_B63_4
ellipse at (283,282)-(294,293): alarm colour if ST03_422_B64_3.BitInToCheck; tooltip ST03_422_B64_3
rounded rectangle at (271,432)-(290,449): alarm colour if ST03_422_B64_4.BitInToCheck; tooltip ST03_422_B64_4
embedded screen at (0,317)-(179,437): ZLIB_SENSOPART_2; invisible if MP.ST02.SensopartEthernet
rectangle at (276,266)-(286,291): invisible if ST03_160pol_Zufuehrung.CamResult < 11; alarm colour if ST03_160pol_Zufuehrung.CamResult = 99
rectangle at (276,267)-(286,293): invisible if ST03_160pol_Zufuehrung.CamResult >= 11 OR NOT ST03_422_B64_3.BitInToCheck
rectangle at (276,391)-(286,437): invisible if NOT ST03_422_B64_4.BitInToCheck; alarm colour if ST03_Main.Result=RESULT_NOK
rectangle at (271,296)-(292,303): alarm colour if ST03_422_B64_1.ValveSensor; tooltip ST03_422_B64_1
rectangle at (271,184)-(292,191): alarm colour if ST03_421_B63_2.ValveSensor; tooltip ST03_421_B63_2
rectangle at (271,140)-(292,147): alarm colour if ST03_421_B63_0.ValveSensor; tooltip ST03_421_B63_0
rectangle at (275,212)-(286,226): alarm colour if ST03_421_B63_7.BitInToCheck
ellipse at (283,171)-(294,182): alarm colour if ST03_421_B63_7.BitInToCheck; tooltip ST03_421_B63_7
rounded rectangle at (292,17)-(303,69): alarm colour if ST03_Init_Lockings.b_freiFuerSG; tooltip b_freiFuerSG
embedded screen at (0,317)-(179,438): ZLIB_SENSOPART_6; invisible if NOT MP.ST02.SensopartEthernet
ellipse at (282,319)-(293,330): alarm colour if ST03_423_B65_2.BitInToCheck; tooltip ST03_423_B65_2
rectangle at (275,305)-(285,330): invisible if ST03_160pol_Zufuehrung.CamResult2 < 11; alarm colour if ST03_160pol_Zufuehrung.CamResult2 = 99
rectangle at (275,306)-(285,331): invisible if ST03_160pol_Zufuehrung.CamResult2 >= 11 OR NOT ST03_423_B65_2.BitInToCheck
rectangle at (271,334)-(292,341): alarm colour if ST03_423_B65_0.ValveSensor; tooltip ST03_423_B65_0
ellipse at (283,355)-(294,366): alarm colour if ST03_423_B65_5.BitInToCheck; tooltip ST03_423_B65_5
rectangle at (276,343)-(286,365): invisible if ST03_160pol_Zufuehrung.CamResult3 < 11; alarm colour if ST03_160pol_Zufuehrung.CamResult3 = 99
rectangle at (276,344)-(286,367): invisible if ST03_160pol_Zufuehrung.CamResult3 >= 11 OR NOT ST03_423_B65_5.BitInToCheck
rectangle at (271,369)-(292,376): alarm colour if ST03_423_B65_4.ValveSensor; tooltip ST03_423_B65_4
rectangle at (187,270)-(264,295): text "%d"; shows NokCounter1li; editable
rectangle at (187,306)-(264,331): text "%d"; shows NokCounter2li; editable
rectangle at (187,344)-(264,369): text "%d"; shows NokCounter3li; editable
rectangle at (296,344)-(373,369): text "%d"; shows NokCounter3re; editable
rectangle at (296,307)-(373,332): text "%d"; shows NokCounter2re; editable
rectangle at (296,269)-(374,294): text "%d"; shows NokCounter1re; editable
rectangle at (299,245)-(374,270): text "%<BASIC>"; shows 'NIO Kamera'
rectangle at (187,246)-(265,271): text "%<BASIC>"; shows 'NIO Kamera'
rounded rectangle at (271,228)-(290,245): alarm colour if ST03_423_B66_0.BitInToCheck; tooltip ST03_423_B66_0
rectangle at (275,232)-(286,246): alarm colour if ST03_421_B63_7.BitInToCheck
rectangle at (167,196)-(254,239): shows 'Tank voll'
rectangle at (182,195)-(233,214): text "%<BASIC>"; shows 'bereit'
ellipse at (237,199)-(248,210): alarm colour if ST03_70U3_1.BitInToCheck
ellipse at (170,200)-(181,211): alarm colour if ST03_71U3_1.BitInToCheck
rectangle at (182,207)-(233,226): text "%<BASIC>"; shows 'Störung'
ellipse at (237,211)-(248,222): invisible if MP.ST03.SGM_3621; alarm colour if ST03_70U3_2.BitInToCheck
ellipse at (170,212)-(181,223): invisible if MP.ST03.SGM_3621; alarm colour if ST03_71U3_2.BitInToCheck
rectangle at (182,219)-(233,238): text "%<BASIC>"; shows 'Störung'
ellipse at (237,223)-(248,234): alarm colour if ST03_70U3_3.BitInToCheck
ellipse at (170,224)-(181,235): alarm colour if ST03_71U3_3.BitInToCheck
rectangle at (167,183)-(254,197): text "%<BASIC>"; shows 'li_Drucker_re'
3 more shapes without text or variables
*)

(* Visualisation ZUFUEHRUNG_191POL
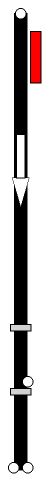
embedded screen at (9,126)-(26,199): SIGNS_ARROWDOWN
ellipse at (12,0)-(23,11): alarm colour if ST03_541_B69_0.BitInToCheck; tooltip ST03_541_B69_0
ellipse at (19,368)-(30,379): alarm colour if ST03_541_B69_6.BitInToCheck; tooltip ST03_541_B69_6
rectangle at (7,380)-(28,387): alarm colour if ST03_541_B69_4.ValveSensor; tooltip ST03_541_B69_3
rectangle at (7,316)-(28,323): alarm colour if ST03_541_B69_2.ValveSensor; tooltip ST03_541_B69_1
rounded rectangle at (27,23)-(38,75): alarm colour if ST03_Init_Lockings.b_freiFuerSG; tooltip b_freiFuerSG
ellipse at (19,454)-(30,465): alarm colour if ST03_542_B70_0.BitInToCheck; tooltip ST03_542_B70_0
ellipse at (5,454)-(16,465): alarm colour if ST03_541_B69_7.BitInToCheck; tooltip ST03_542_B70_0
2 more shapes without text or variables
*)

(* Visualisation ZUFUEHRUNG_206POL
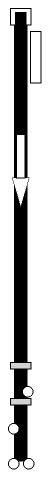
ellipse at (30,455)-(41,466): alarm colour if ST03_436_B68_1.BitInToCheck; tooltip ST03_436_B68_1
embedded screen at (19,131)-(36,204): SIGNS_ARROWDOWN
ellipse at (15,455)-(26,466): alarm colour if ST03_436_B68_2.BitInToCheck; tooltip ST03_436_B68_2
ellipse at (15,420)-(26,431): alarm colour if ST03_437_B68_4.BitInToCheck; tooltip ST03_437_B68_4
ellipse at (29,383)-(40,394): alarm colour if ST03_435_B67_7.BitInToCheck; tooltip ST03_435_B67_7
rectangle at (17,395)-(38,402): alarm colour if .ST03_435_B67_2.ValveSensor; tooltip .ST03_435_B67_2
rectangle at (17,359)-(38,366): alarm colour if ST03_435_B67_1.ValveSensor; tooltip ST03_435_B67_1
rounded rectangle at (17,5)-(38,22): alarm colour if ST03_435_B67_4.BitInToCheck; tooltip ST03_435_B67_4
rounded rectangle at (37,28)-(48,80): alarm colour if ST03_Init_Lockings.b_freiFuerSG; tooltip b_freiFuerSG
2 more shapes without text or variables
*)

(* Visualisation ZUFUEHRUNG_21POL
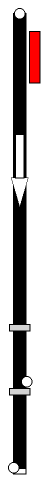
embedded screen at (9,126)-(26,199): SIGNS_ARROWDOWN
ellipse at (12,0)-(23,11): alarm colour if ST03_536_B69_0.BitInToCheck; tooltip ST03_536_B69_0
ellipse at (19,368)-(30,379): alarm colour if ST03_536_B69_6.BitInToCheck; tooltip ST03_536_B69_6
rectangle at (7,380)-(28,387): alarm colour if ST03_536_B69_4.ValveSensor; tooltip ST03_536_B69_3
rectangle at (7,316)-(28,323): alarm colour if ST03_536_B69_2.ValveSensor; tooltip ST03_536_B69_1
rounded rectangle at (27,23)-(38,75): alarm colour if ST03_Init_Lockings.b_freiFuerSG; tooltip b_freiFuerSG
rectangle at (11,460)-(24,466): alarm colour if ST03_537_B70_0.BitInToCheck; tooltip ST03_537_B70_0
ellipse at (6,454)-(17,465): alarm colour if ST03_536_B69_7.BitInToCheck; tooltip ST03_536_B69_7
2 more shapes without text or variables
*)

(* Visualisation ZUFUEHRUNG_268POL_102POL_NEU
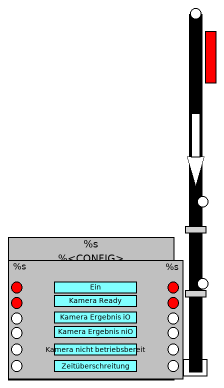
embedded screen at (179,202)-(196,275): SIGNS_ARROWDOWN
ellipse at (182,97)-(193,108): alarm colour if ST03_556_B69_0.BitInToCheck; tooltip ST03_556_B69_0
ellipse at (189,367)-(200,378): alarm colour if ST03_556_B69_6.BitInToCheck; tooltip ST03_556_B69_6
rectangle at (177,379)-(198,386): alarm colour if ST03_556_B69_4.ValveSensor; tooltip ST03_541_B69_3
rectangle at (177,315)-(198,322): alarm colour if ST03_556_B69_2.ValveSensor; tooltip ST03_541_B69_1
rounded rectangle at (175,448)-(199,465): alarm colour if ST03_556_B69_7.BitInToCheck; tooltip ST03_556_B69_7
rounded rectangle at (197,120)-(208,172): alarm colour if ST03_Init_Lockings.b_freiFuerSG; tooltip b_freiFuerSG
ellipse at (189,285)-(200,296): alarm colour if ST03_556_B69_5.BitInToCheck; tooltip ST03_556_B69_5
embedded screen at (0,326)-(166,469): ZLIB_SENSOPART_5; invisible if gTypeCode <> 5841
embedded screen at (0,349)-(175,468): ZLIB_SENSOPART_6; invisible if gTypeCode <> 4993
2 more shapes without text or variables
*)

(* Visualisation ZUFUEHRUNG_268POL_RP
